INTERFACE Drive

END_INTERFACE

(* stored: Version 1.1.0.1, ProductVersion 3.1.4024.11
   Itf Drive: Id {0480bdaa-c1a1-44cb-8ff4-3560f0f2fc6e} *)
